FUNCTION_BLOCK A2X2_CLIENT_2_0_SUBSCRIBE_2_PLUG (* Write both BOOLs of an A2X2 adapter as a remote OPC-UA write via CLIENT_2_0 and read both back via SUBSCRIBE_2, driven by an A2X2 bidirectional adapter Plug (mirror of A2X2_CLIENT_2_0_SUBSCRIBE_2, which uses a Socket), each BOOL buffered with its own E_D_FF *)
  (* Standard: 61499-2; Description: Copyright (c) 2026 HR Agrartechnik GmbH This program and the accompanying materials are made available under the terms of the Eclipse Public License 2.0 which is available at https://www.eclipse.org/legal/epl-2.0/ SPDX-License-Identifier: EPL-2.0 *)
  (* Version 1.0, 2026-09-05, Franz Höpfinger, HR Agrartechnik GmbH, initial API and implementation and/or initial documentation *)
  PACKAGE adapter::net;
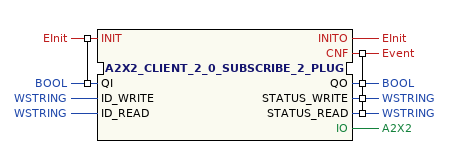
  EVENT_INPUT
    INIT : EInit WITH QI; (* Initialization *)
  END_EVENT
  EVENT_OUTPUT
    INITO : EInit; (* Initialization Confirm *)
    CNF WITH QO, STATUS_WRITE, STATUS_READ; (* QO/STATUS updated *)
  END_EVENT
  VAR_INPUT
    QI : BOOL;
    ID_WRITE : WSTRING; (* Remote-Zieladresse (ACTION=WRITE) fuer beide BOOLs *)
    ID_READ : WSTRING; (* Lokal ueberwachter Zustandsknoten (ACTION=READ) fuer beide BOOLs *)
  END_VAR
  VAR_OUTPUT
    QO : BOOL; (* TRUE nur wenn WRITE_CLIENT und READ_SUBSCRIBE aktuell beide QO=TRUE melden *)
    STATUS_WRITE : WSTRING; (* STATUS von WRITE_CLIENT *)
    STATUS_READ : WSTRING; (* STATUS von READ_SUBSCRIBE *)
  END_VAR
  PLUGS
    IO : adapter::types::bidirectional::A2X2; (* UP/DOWN BOOLs to send (out), UP/DOWN BOOLs received (in) *)
  END_PLUGS
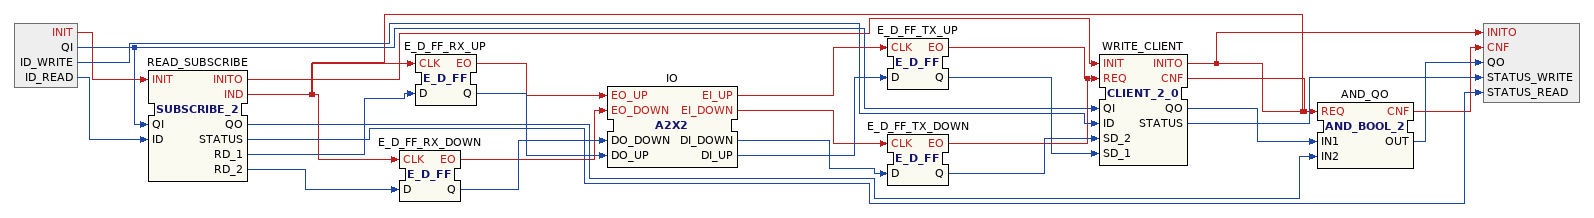
  FBS
    WRITE_CLIENT : iec61499::net::CLIENT_2_0;
    READ_SUBSCRIBE : iec61499::net::SUBSCRIBE_2;
    AND_QO : iec61131::booleanOperators::AND_BOOL_2;
    E_D_FF_RX_UP : iec61499::events::E_D_FF;
    E_D_FF_RX_DOWN : iec61499::events::E_D_FF;
    E_D_FF_TX_UP : iec61499::events::E_D_FF;
    E_D_FF_TX_DOWN : iec61499::events::E_D_FF;
  END_FBS
  EVENT_CONNECTIONS
    INIT TO READ_SUBSCRIBE.INIT;
    READ_SUBSCRIBE.INITO TO WRITE_CLIENT.INIT;
    WRITE_CLIENT.INITO TO INITO;
    WRITE_CLIENT.INITO TO AND_QO.REQ;
    WRITE_CLIENT.CNF TO AND_QO.REQ;
    READ_SUBSCRIBE.IND TO AND_QO.REQ;
    AND_QO.CNF TO CNF;
    READ_SUBSCRIBE.IND TO E_D_FF_RX_UP.CLK;
    READ_SUBSCRIBE.IND TO E_D_FF_RX_DOWN.CLK;
    E_D_FF_RX_UP.EO TO IO.EO_UP;
    E_D_FF_RX_DOWN.EO TO IO.EO_DOWN;
    IO.EI_UP TO E_D_FF_TX_UP.CLK;
    IO.EI_DOWN TO E_D_FF_TX_DOWN.CLK;
    E_D_FF_TX_DOWN.EO TO WRITE_CLIENT.REQ;
    E_D_FF_TX_UP.EO TO WRITE_CLIENT.REQ;
  END_CONNECTIONS
  DATA_CONNECTIONS
    QI TO READ_SUBSCRIBE.QI;
    QI TO WRITE_CLIENT.QI;
    ID_READ TO READ_SUBSCRIBE.ID;
    ID_WRITE TO WRITE_CLIENT.ID;
    WRITE_CLIENT.QO TO AND_QO.IN1;
    READ_SUBSCRIBE.QO TO AND_QO.IN2;
    AND_QO.OUT TO QO;
    WRITE_CLIENT.STATUS TO STATUS_WRITE;
    READ_SUBSCRIBE.STATUS TO STATUS_READ;
    READ_SUBSCRIBE.RD_1 TO E_D_FF_RX_UP.D;
    READ_SUBSCRIBE.RD_2 TO E_D_FF_RX_DOWN.D;
    E_D_FF_RX_DOWN.Q TO IO.DO_DOWN;
    E_D_FF_RX_UP.Q TO IO.DO_UP;
    IO.DI_DOWN TO E_D_FF_TX_DOWN.D;
    IO.DI_UP TO E_D_FF_TX_UP.D;
    E_D_FF_TX_DOWN.Q TO WRITE_CLIENT.SD_2;
    E_D_FF_TX_UP.Q TO WRITE_CLIENT.SD_1;
  END_CONNECTIONS
END_FUNCTION_BLOCK
